// TIA Portal V16 export
// export: Created 2021-11-12T13:32:33.46356Z, ExportSetting WithDefaults, DisplayName Totally Integrated Automation Portal, DisplayVersion V16 Update 3, DisplayName TIA Portal Version Control Interface, DisplayVersion V16 Update 2, DisplayName TIA Portal Openness, DisplayVersion V16 Update 3, DisplayName SINAMICS Startdrive Advanced, DisplayVersion V16 Update 5, DisplayName SINAMICS Startdrive G130, G150, S120, S150, SINAMICS MV, S210, DisplayVersion V16 Update 5, DisplayName SINAMICS Startdrive G110M, G120, G120C, G120D, G120P, G115D, DisplayVersion V16 Update 5, DisplayName STEP 7 Professional, DisplayVersion V16 Update 3, DisplayName STEP 7 Safety, DisplayVersion V16, DisplayName WinCC UA Professional, DisplayVersion V16 Update 3
DATA_BLOCK "IDB_Zone100"   // DB16
{ DB_Accessible_From_OPC_UA := 'FALSE' }
VERSION : 0.1
// stored: AutoNumber true, DBAccessibleFromOPCUA false, InstanceOfName Zone100, InstanceOfType FB
"Zone100"
   // VAR
   //    SF_ZoneMode { S7_SetPoint := 'True'} : "STD_Zone";
   //    SF_StationKAS1Mode { S7_SetPoint := 'True'} : "STD_Station";
   //    SF_StationKAS2Mode { S7_SetPoint := 'True'} : "STD_Station";
   //    SF_Station110Mode { S7_SetPoint := 'True'} : "STD_Station";
   //    SF_Station120Mode { S7_SetPoint := 'True'} : "STD_Station";
   //    SF_Station1R1Mode { S7_SetPoint := 'True'} : "STD_Station";
   //    SF_Station1R2Mode { S7_SetPoint := 'True'} : "STD_Station";
   //    SF_Station130Mode { S7_SetPoint := 'True'} : "STD_Station";
   //    SF_Station140Mode { S7_SetPoint := 'True'} : "STD_Station";
   //    SF_Station1R3Mode { S7_SetPoint := 'True'} : "STD_Station";
   //    SF_Station1R4Mode { S7_SetPoint := 'True'} : "STD_Station";
   //    SF_Station150Mode { S7_SetPoint := 'True'} : "STD_Station";
   //    SF_Station160Mode { S7_SetPoint := 'True'} : "STD_Station";
   //    SF_Station170Mode { S7_SetPoint := 'True'} : "STD_Station";
   //    SF_Station180Mode { S7_SetPoint := 'True'} : "STD_Station";
   //    SF_Station1R5Mode { S7_SetPoint := 'True'} : "STD_Station";
   //    SF_Station1R6Mode { S7_SetPoint := 'True'} : "STD_Station";
   //    SF_StationBSN1Mode { S7_SetPoint := 'True'} : "STD_Station";
   //    SF_StationBSN2Mode { S7_SetPoint := 'True'} : "STD_Station";
   //    SF_CameraLights { S7_SetPoint := 'True'} : "STD_OnOff";
   //    ST_TONZone1ServModeAct { S7_SetPoint := 'True'} : TON_TIME;
   //    SS_Edge { S7_SetPoint := 'True'} : Array[0..100] of Bool;
   // END_VAR
BEGIN
END_DATA_BLOCK
